{attribute 'qualified_only'}
VAR_GLOBAL PERSISTENT
	stLogDemo  : ST_MbLog;
	stLogMeter : ST_MbLog;
END_VAR

(* stored: Version 1.1.0.1
   GVL GVL_Log: Id {6fad0097-072c-429f-bff2-db002af7e598} *)
